// TIA Portal V19 export
TYPE "LAF_typeAxisDiagErrorDetail"
TITLE = LAF_typeAxisDiagErrorDetail
// Alarm number and effective alarm response of a Technology Object
// stored: Access Published
   STRUCT
      number { ExternalWritable := 'False'} : UDInt;   // Alarm number
      reaction { ExternalWritable := 'False'} : DInt;   // Effective alarm response (0=no reaction, 1=stop with current dynamic values, 2=stop with maximum dynamic values, 3=stop with emergency stop ramp, 4=remove enable, 5=track setpoints); external encoder (0=no reaction, 10=remove enable)
   END_STRUCT;
END_TYPE
